(* LS Electric XG5000 project: test *)
(* PLC LSPLC *)

FUNCTION 시간검출 : ARRAY[0..5] OF WORD
VAR_INPUT
    _RTC_TIME_0 : BYTE;
    _RTC_TIME_1 : BYTE;
    _RTC_TIME_2 : BYTE;
    _RTC_TIME_3 : BYTE;
    _RTC_TIME_4 : BYTE;
    _RTC_TIME_5 : BYTE;
END_VAR

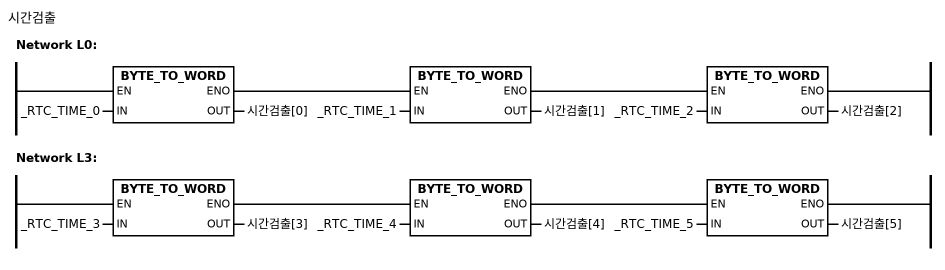
(* Rung L0 *)
시간검출[0] := BYTE_TO_WORD(_RTC_TIME_0);
시간검출[1] := BYTE_TO_WORD(_RTC_TIME_1);
시간검출[2] := BYTE_TO_WORD(_RTC_TIME_2);
(* Rung L3 *)
시간검출[3] := BYTE_TO_WORD(_RTC_TIME_3);
시간검출[4] := BYTE_TO_WORD(_RTC_TIME_4);
시간검출[5] := BYTE_TO_WORD(_RTC_TIME_5);
END_FUNCTION

FUNCTION_BLOCK 사칙연산산
VAR_INPUT
    in1 : REAL;
    in2 : REAL;
END_VAR
VAR_OUTPUT
    addOut : REAL;
    subOut : REAL;
    mulOut : REAL;
    divOut : REAL;
END_VAR

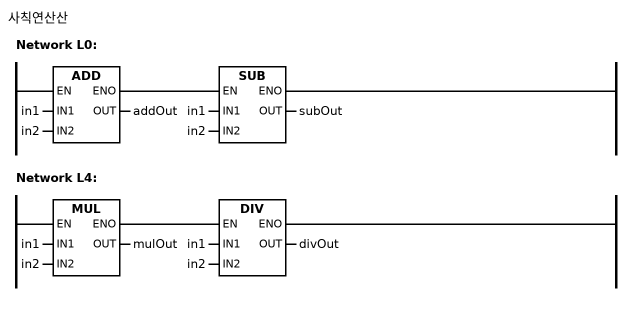
(* Rung L0 *)
addOut := in1 + in2;
subOut := in1 - in2;
(* Rung L4 *)
mulOut := in1 * in2;
divOut := in1 / in2;
END_FUNCTION_BLOCK

FUNCTION_BLOCK PITA
VAR_INPUT
    A변 : REAL;
    B변 : REAL;
END_VAR
VAR_OUTPUT
    Result : REAL;
END_VAR
VAR
    A제곱 : REAL;
    A제쁠B제 : REAL;
    B제곱 : REAL;
END_VAR

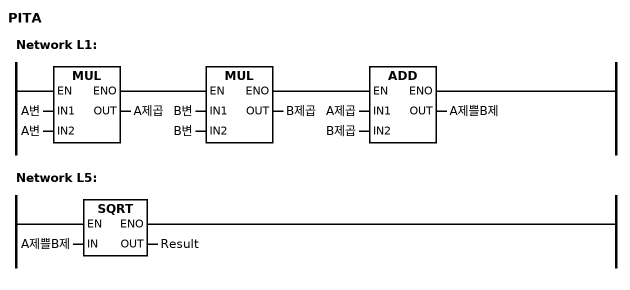
(* Rung L1 *)
A제곱 := A변 * A변;
B제곱 := B변 * B변;
A제쁠B제 := A제곱 + B제곱;
(* Rung L5 *)
Result := SQRT(A제쁠B제);
END_FUNCTION_BLOCK

FUNCTION_BLOCK 깜빡이
VAR_INPUT
    FL : BOOL;
    NFL : BOOL;
    OFF : BOOL;
END_VAR
VAR_OUTPUT
    LA1 : BOOL;
    LA2 : BOOL;
END_VAR
VAR
    T1 : TON;
    T2 : TON;
    T3 : TON;
    temp : BOOL;
    tp1 : TP;
END_VAR

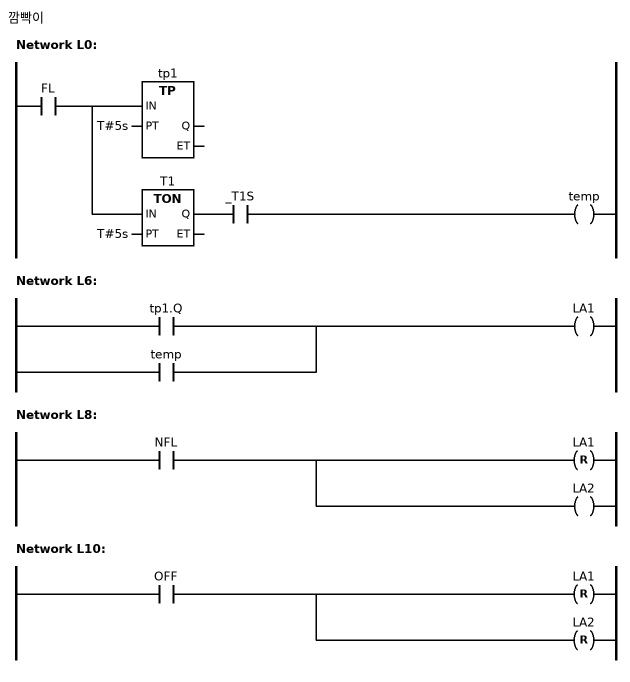
(* Rung L0 *)
tp1(IN := FL, PT := T#5s);
T1(IN := FL, PT := T#5s);
temp := T1.Q AND _T1S;
(* Rung L6 *)
LA1 := tp1.Q OR temp;
(* Rung L8 *)
IF NFL THEN LA1 := FALSE; END_IF;
LA2 := NFL;
(* Rung L10 *)
IF OFF THEN
    LA1 := FALSE;
    LA2 := FALSE;
END_IF;
END_FUNCTION_BLOCK

PROGRAM 1stDay (* task: 스캔 프로그램 *)
VAR
    addOut : BOOL;
    in1 : BOOL;
    in2 : BOOL;
    in3 : BOOL;
    in4 : BOOL;
    INST : TON;
    int1 : INT;
    int2 : INT;
    int3 : INT;
    out1 : BOOL;
    out2 : BOOL;
    out3 : BOOL;
    out4 : BOOL;
    PB0 : BOOL;
    PB1 : BOOL;
    time1 : TIME;
    time2 : TIME;
    timeOut : BOOL;
    램프 : BOOL;
    모터1 : BOOL;
    모터2 : BOOL;
    모터3 : BOOL;
    스위치 : BOOL;
    펄스 : BOOL;
END_VAR
VAR
    _e1 : R_TRIG;
    _e2 : R_TRIG;
    _e3 : R_TRIG;
    _e4 : R_TRIG;
    _e5 : R_TRIG;
    _e6 : R_TRIG;
    _e7 : R_TRIG;
END_VAR

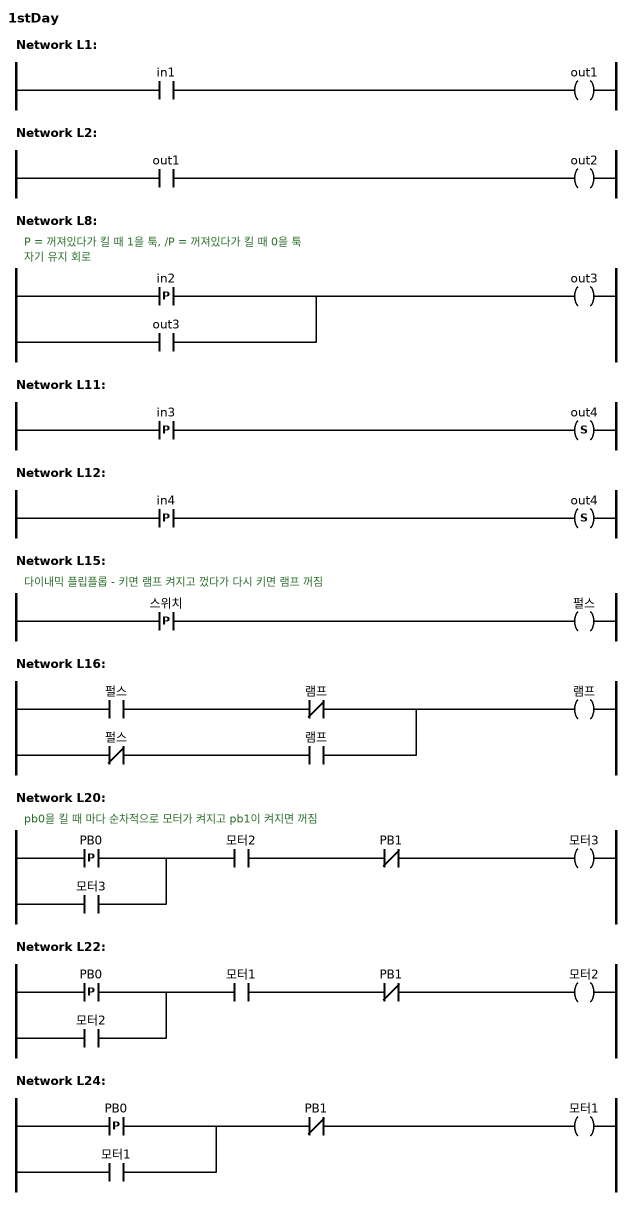
(* Rung L1 *)
out1 := in1;
(* Rung L2 *)
out2 := out1;
(* P = 꺼져있다가 킬 때 1을 툭, /P = 꺼져있다가 킬 때 0을 툭 *)
(* 자기 유지 회로 *)
(* Rung L8 *)
_e1(CLK := in2);
out3 := _e1.Q OR out3;
(* Rung L11 *)
_e2(CLK := in3);
IF _e2.Q THEN out4 := TRUE; END_IF;
(* Rung L12 *)
_e3(CLK := in4);
IF _e3.Q THEN out4 := TRUE; END_IF;
(* 다이내믹 플립플롭 - 키면 램프 켜지고 껐다가 다시 키면 램프 꺼짐 *)
(* Rung L15 *)
_e4(CLK := 스위치);
펄스 := _e4.Q;
(* Rung L16 *)
램프 := (펄스 AND NOT 램프) OR (NOT 펄스 AND 램프);
(* pb0을 킬 때 마다 순차적으로 모터가 켜지고 pb1이 켜지면 꺼짐 *)
(* Rung L20 *)
_e5(CLK := PB0);
모터3 := (_e5.Q OR 모터3) AND 모터2 AND NOT PB1;
(* Rung L22 *)
_e6(CLK := PB0);
모터2 := (_e6.Q OR 모터2) AND 모터1 AND NOT PB1;
(* Rung L24 *)
_e7(CLK := PB0);
모터1 := (_e7.Q OR 모터1) AND NOT PB1;
END_PROGRAM

PROGRAM 2ndDay (* task: 스캔 프로그램 *)
VAR
    addOut : BOOL;
    in1 : BOOL;
    in2 : BOOL;
    in3 : BOOL;
    INST : TON;
    INST1 : TP;
    int1 : INT;
    int2 : INT;
    int3 : INT;
    moveIn : INT;
    moveOut : INT;
    out1 : BOOL;
    out2 : BOOL;
    out3 : BOOL;
    out4 : BOOL;
    T4 : TON;
    T4_스위치 : BOOL;
    T5 : TON;
    T6 : TON;
    T7 : TOF;
    T8 : TOF;
    time1 : TIME;
    time2 : TIME;
    timeOut : BOOL;
    trigger : BOOL;
    결과1 : INT;
    결과1_R : REAL;
    꺼져있는시간 : TIME;
    나가면물 : TP;
    나가면물켜 : TON_UINT;
    년출력 : WORD;
    대기 : TON;
    대기시간 : TIME;
    들어오면물 : TP;
    램프 : BOOL;
    램프4 : BOOL;
    물 : TP;
    물끔대기 : TOF;
    물켜 : TON;
    숫자1 : INT;
    숫자1_R : REAL;
    스위치 : BOOL;
    시간검출배열 : ARRAY[0..5] OF WORD;
    월출력 : WORD;
    이탈하면물 : TP;
    일출력 : WORD;
    접근 : BOOL;
    접근하면물 : TP;
    카운트업 : CTU_INT;
    카운트업리셋 : BOOL;
    카운트업스위치 : BOOL;
    켜져있는시간 : TIME;
    콸콸콸 : BOOL;
END_VAR

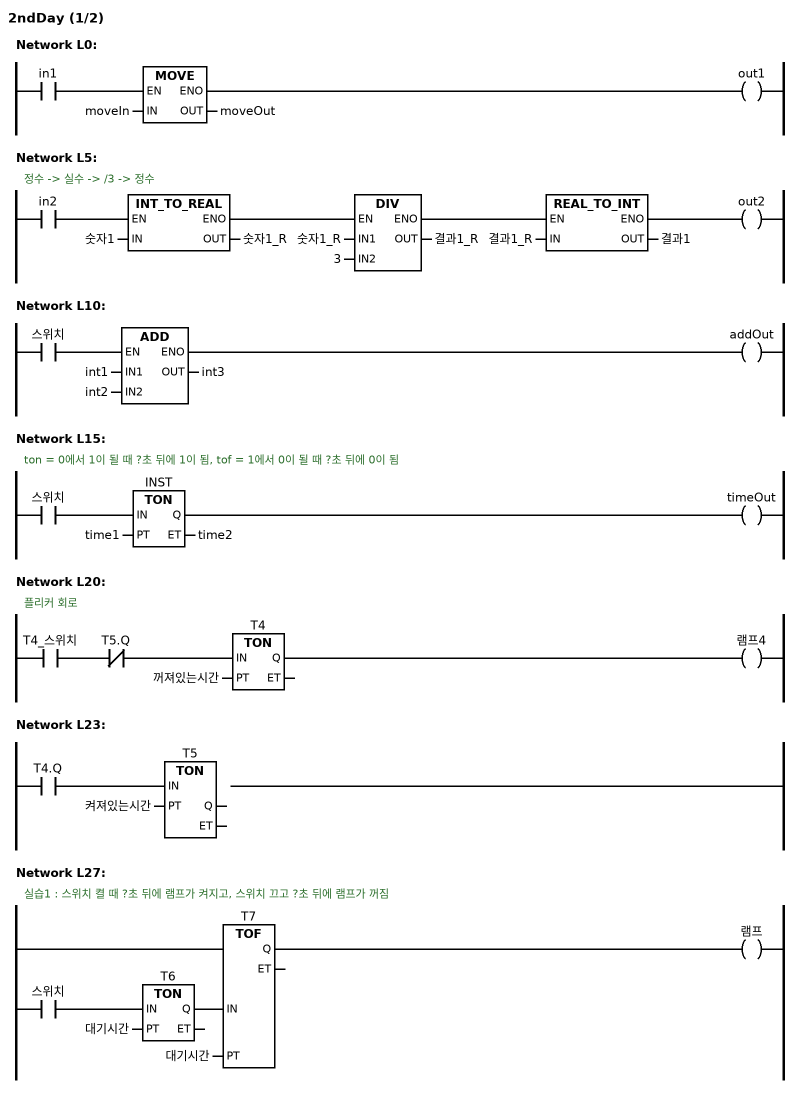
(* Rung L0 *)
IF in1 THEN moveOut := moveIn; END_IF;
out1 := in1;
(* 정수 -> 실수 -> /3 -> 정수 *)
(* Rung L5 *)
IF in2 THEN
    숫자1_R := INT_TO_REAL(숫자1);
    결과1_R := 숫자1_R / 3;
    결과1 := REAL_TO_INT(결과1_R);
END_IF;
out2 := in2;
(* Rung L10 *)
IF 스위치 THEN int3 := int1 + int2; END_IF;
addOut := 스위치;
(* ton = 0에서 1이 될 때 ?초 뒤에 1이 됨, tof = 1에서 0이 될 때 ?초 뒤에 0이 됨 *)
(* Rung L15 *)
INST(IN := 스위치, PT := time1, ET => time2);
timeOut := INST.Q;
(* 플리커 회로 *)
(* Rung L20 *)
T4(IN := T4_스위치 AND NOT T5.Q, PT := 꺼져있는시간);
램프4 := T4.Q;
(* Rung L23 *)
T5(IN := T4.Q, PT := 켜져있는시간);
(* 실습1 : 스위치 켤 때 ?초 뒤에 램프가 켜지고, 스위치 끄고 ?초 뒤에 램프가 꺼짐 *)
(* Rung L27 *)
T6(IN := 스위치, PT := 대기시간);
T7(IN := T6.Q, PT := 대기시간);
램프 := T7.Q;

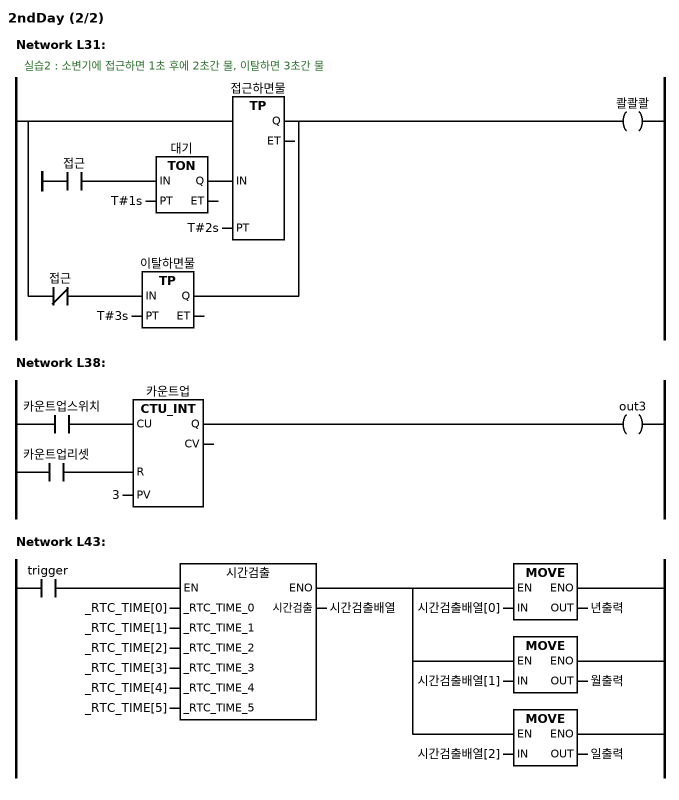
(* 실습2 : 소변기에 접근하면 1초 후에 2초간 물, 이탈하면 3초간 물 *)
(* Rung L31 *)
대기(IN := 접근, PT := T#1s);
접근하면물(IN := 대기.Q, PT := T#2s);
이탈하면물(IN := NOT 접근, PT := T#3s);
콸콸콸 := 접근하면물.Q OR 이탈하면물.Q;
(* Rung L38 *)
카운트업(CU := 카운트업스위치, R := 카운트업리셋, PV := 3);
out3 := 카운트업.Q;
(* Rung L43 *)
IF trigger THEN
    시간검출배열 := 시간검출(_RTC_TIME_0 := _RTC_TIME[0], _RTC_TIME_1 := _RTC_TIME[1], _RTC_TIME_2 := _RTC_TIME[2], _RTC_TIME_3 := _RTC_TIME[3], _RTC_TIME_4 := _RTC_TIME[4], _RTC_TIME_5 := _RTC_TIME[5]);
    년출력 := 시간검출배열[0];
    월출력 := 시간검출배열[1];
    일출력 := 시간검출배열[2];
END_IF;
END_PROGRAM

PROGRAM 3rdDay (* task: 스캔 프로그램 *)
VAR
    a : REAL;
    addOut : REAL;
    b : REAL;
    divOut : REAL;
    FL : BOOL;
    LA1 : BOOL;
    LA2 : BOOL;
    mulOut : REAL;
    NFL : BOOL;
    OFF : BOOL;
    out1 : BOOL;
    out2 : BOOL;
    p0 : BOOL;
    p1 : BOOL;
    p10 : BOOL;
    p11 : BOOL;
    p2 : BOOL;
    p3 : BOOL;
    pOut : BOOL;
    subOut : REAL;
    t0 : TON;
    t1 : TON;
    계산기 : 사칙연산산;
    램 : BOOL;
    램프 : 깜빡이;
    램프1 : BOOL;
    램프2 : BOOL;
    피타고라스의정의 : PITA;
END_VAR

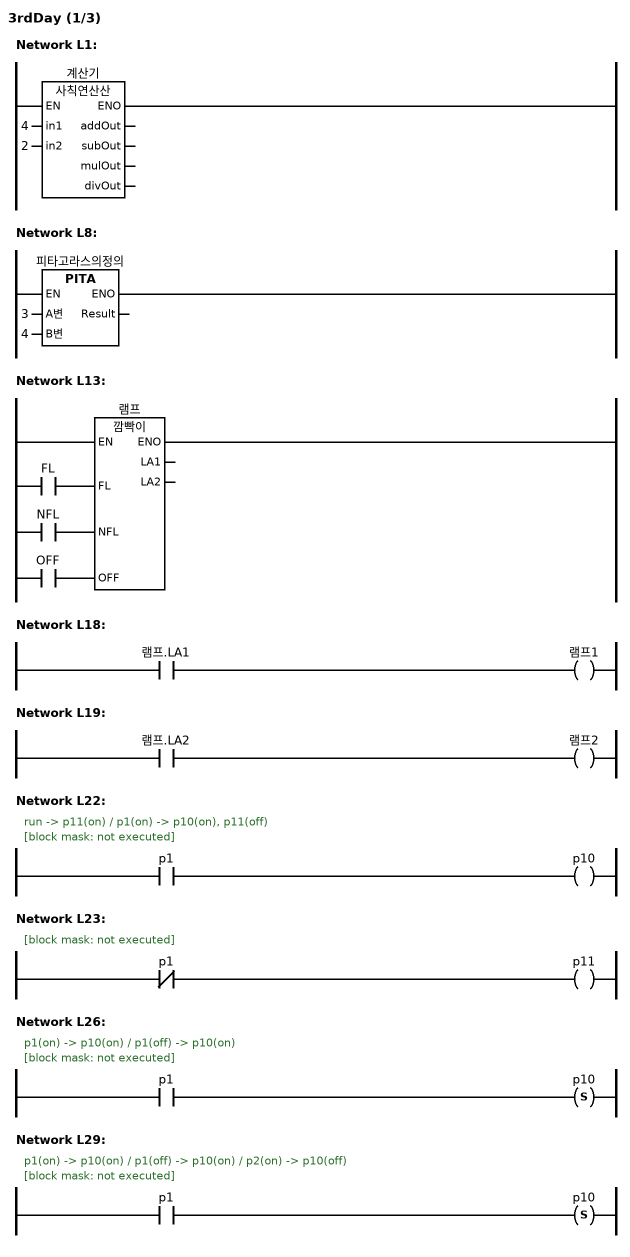
(* Rung L1 *)
계산기(in1 := 4, in2 := 2);
(* Rung L8 *)
피타고라스의정의(A변 := 3, B변 := 4);
(* Rung L13 *)
램프(FL := FL, NFL := NFL, OFF := OFF);
(* Rung L18 *)
램프1 := 램프.LA1;
(* Rung L19 *)
램프2 := 램프.LA2;
(* run -> p11(on) / p1(on) -> p10(on), p11(off) *)
(* Rung L22 is block-masked: not executed *)
// p10 := p1;
(* Rung L23 is block-masked: not executed *)
// p11 := NOT p1;
(* p1(on) -> p10(on) / p1(off) -> p10(on) *)
(* Rung L26 is block-masked: not executed *)
// IF p1 THEN p10 := TRUE; END_IF;
(* p1(on) -> p10(on) / p1(off) -> p10(on) / p2(on) -> p10(off) *)
(* Rung L29 is block-masked: not executed *)
// IF p1 THEN p10 := TRUE; END_IF;

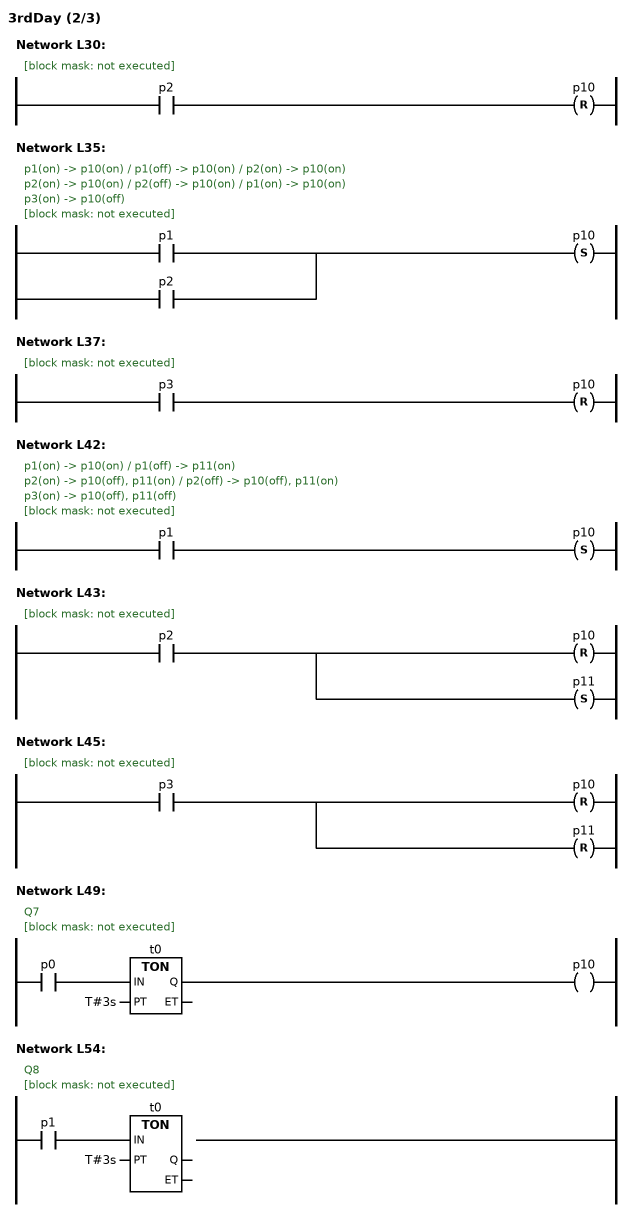
(* Rung L30 is block-masked: not executed *)
// IF p2 THEN p10 := FALSE; END_IF;
(* p1(on) -> p10(on) / p1(off) -> p10(on) / p2(on) -> p10(on) *)
(* p2(on) -> p10(on) / p2(off) -> p10(on) / p1(on) -> p10(on) *)
(* p3(on) -> p10(off) *)
(* Rung L35 is block-masked: not executed *)
// IF p1 OR p2 THEN p10 := TRUE; END_IF;
(* Rung L37 is block-masked: not executed *)
// IF p3 THEN p10 := FALSE; END_IF;
(* p1(on) -> p10(on) / p1(off) -> p11(on) *)
(* p2(on) -> p10(off), p11(on) / p2(off) -> p10(off), p11(on) *)
(* p3(on) -> p10(off), p11(off) *)
(* Rung L42 is block-masked: not executed *)
// IF p1 THEN p10 := TRUE; END_IF;
(* Rung L43 is block-masked: not executed *)
// IF p2 THEN
//     p10 := FALSE;
//     p11 := TRUE;
// END_IF;
(* Rung L45 is block-masked: not executed *)
// IF p3 THEN
//     p10 := FALSE;
//     p11 := FALSE;
// END_IF;
(* Q7 *)
(* Rung L49 is block-masked: not executed *)
// t0(IN := p0, PT := T#3s);
// p10 := t0.Q;
(* Q8 *)
(* Rung L54 is block-masked: not executed *)
// t0(IN := p1, PT := T#3s);

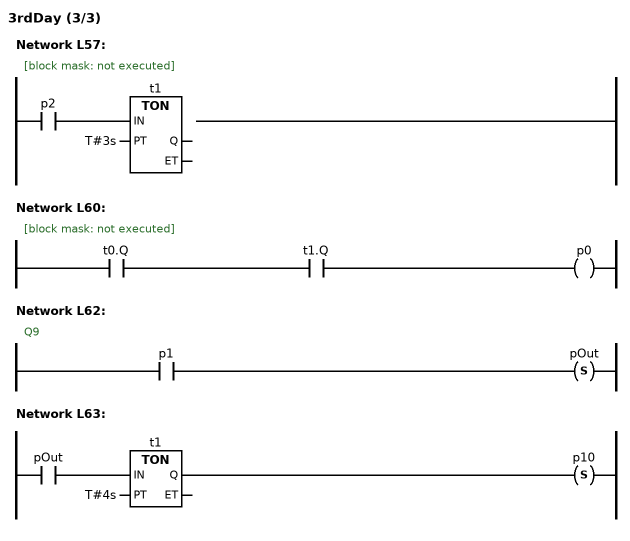
(* Rung L57 is block-masked: not executed *)
// t1(IN := p2, PT := T#3s);
(* Rung L60 is block-masked: not executed *)
// p0 := t0.Q AND t1.Q;
(* Q9 *)
(* Rung L62 *)
IF p1 THEN pOut := TRUE; END_IF;
(* Rung L63 *)
t1(IN := pOut, PT := T#4s);
IF t1.Q THEN p10 := TRUE; END_IF;
END_PROGRAM